FUNCTION_BLOCK FB_Module01 EXTENDS OOP_PackML_Base.FB_Component
VAR_INPUT
END_VAR
VAR_OUTPUT
END_VAR
VAR
	fbLogger:					FB_Logger;
	fbComponent1:				FB_Component;
	fbComponent2:				FB_Component;
	fbComponent3:				FB_Component;
	fbComponent4:				FB_Component;
	bEvent: 					BOOL;
END_VAR

SUPER^();

fbComponent1();
fbComponent2();
fbComponent3();
fbComponent4();

IF bEvent THEN
	bEvent:= FALSE;
	fbComponent1.fbEvent.M_Add('Test');
	fbComponent1.fbEvent.M_Add('Test2');
	fbComponent1.fbEvent.M_Add('Test3');
	fbComponent1.fbEvent.M_Abort('First Error Abort',1);
END_IF

METHOD PROTECTED M_Completing : BOOL
VAR_INPUT
END_VAR
VAR
	nIndex:					DINT;
END_VAR
M_Completing:= TRUE;
WHILE nIndex < fbEvent.fbObserver.nLength DO
	fbEvent.fbObserver.M_Index(nIndex).M_Request(E_Request.Complete);
	nIndex:= nIndex +1;
END_WHILE
END_METHOD

METHOD PROTECTED M_Resetting : BOOL
VAR_INPUT
END_VAR
VAR
	nIndex:					DINT;
END_VAR
M_Resetting:= TRUE;
fbLogger.M_Reset();
WHILE nIndex < fbEvent.fbObserver.nLength DO
	fbEvent.fbObserver.M_Index(nIndex).M_Request(E_Request.Reset);
	nIndex:= nIndex +1;
END_WHILE
END_METHOD

METHOD PROTECTED M_Starting : BOOL
VAR_INPUT
END_VAR
VAR
	nIndex:					DINT;
END_VAR
M_Starting:= TRUE;
WHILE nIndex < fbEvent.fbObserver.nLength DO
	fbEvent.fbObserver.M_Index(nIndex).M_Request(E_Request.Start);
	nIndex:= nIndex +1;
END_WHILE
END_METHOD

METHOD PROTECTED M_Undefined : BOOL;
VAR_INPUT
END_VAR
VAR
	
	nIndex: INT;
END_VAR
IF SUPER^.M_Undefined() THEN
	fbComponent1.fbEvent.P_Logger:= fbLogger;
	fbComponent1.fbEvent.fbObserver.M_Attach(THIS^);
	fbEvent.fbObserver.M_Attach(fbComponent1);
	
	fbComponent2.fbEvent.P_Logger:= fbLogger;
	fbComponent2.fbEvent.fbObserver.M_Attach(THIS^);
	fbEvent.fbObserver.M_Attach(fbComponent2);
	
	fbComponent3.fbEvent.P_Logger:= fbLogger;
	fbComponent3.fbEvent.fbObserver.M_Attach(THIS^);
	fbEvent.fbObserver.M_Attach(fbComponent3);
	
	fbComponent4.fbEvent.P_Logger:= fbLogger;
	fbComponent4.fbEvent.fbObserver.M_Attach(THIS^);
	fbEvent.fbObserver.M_Attach(fbComponent4);
	M_Undefined:= TRUE;
END_IF
END_METHOD

END_FUNCTION_BLOCK

(* stored: Version 1.1.0.1, ProductVersion 3.1.4024.12
   POU FB_Module01: Id {3744d03d-359c-4ab8-84fb-4ea93b7a5162}, SpecialFunc None
   Method M_Completing: Id {38cad43c-ba90-4a92-8ce8-4a165e99aae0}
   Method M_Resetting: Id {fa00b107-60e3-427f-9569-a0a34888482b}
   Method M_Starting: Id {12752945-7cd6-464f-965a-f81c0b828bfd}
   Method M_Undefined: Id {714c485c-83a6-4af2-a706-fec3f6b598e5} *)
